// LS Electric XG5000 project: PLC_222
// PLC LSPLC
// module base 0 slot 0: Input/Output Module:XBC-DR30S (DC 24V Input 18 Contacts, Relay Output 12 Contacts)
// module base 0 slot 9: Analog Input Module:XBO-AD02A (A/D Voltage/Current Input Type(2 Channels))
// module base 0 slot 10: Analog Input Module:XBO-AD02A (A/D Voltage/Current Input Type(2 Channels))

PROGRAM NewProgram (task: Scan Program)

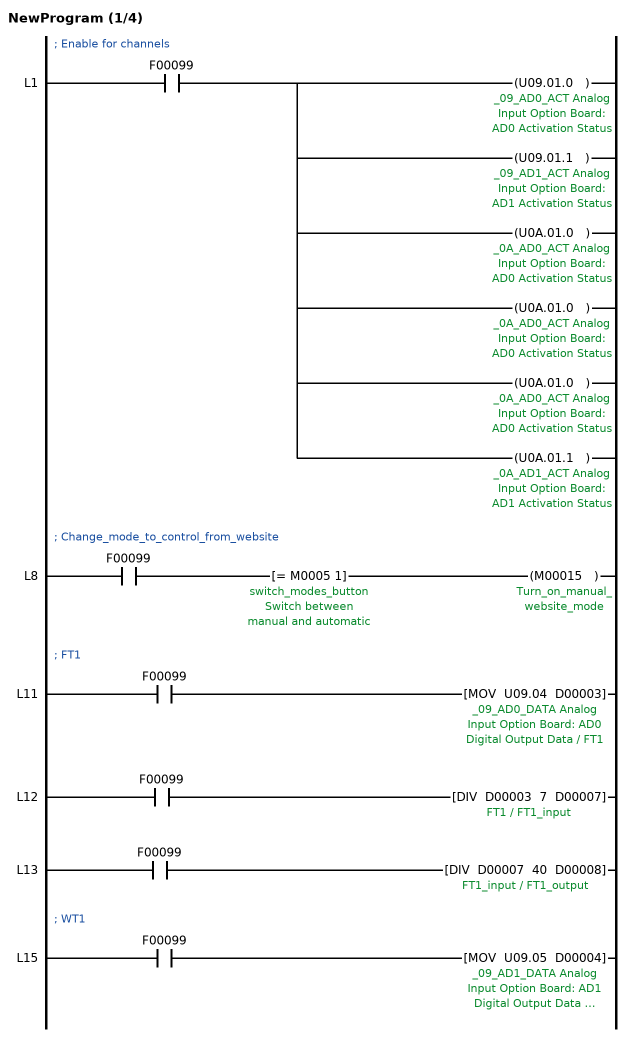
// Enable for channels
; L1
LOAD      F00099
OUT       U09.01.0	// _09_AD0_ACT Analog Input Option Board: AD0 Activation Status
OUT       U09.01.1	// _09_AD1_ACT Analog Input Option Board: AD1 Activation Status
OUT       U0A.01.0	// _0A_AD0_ACT Analog Input Option Board: AD0 Activation Status
OUT       U0A.01.0	// _0A_AD0_ACT Analog Input Option Board: AD0 Activation Status
OUT       U0A.01.0	// _0A_AD0_ACT Analog Input Option Board: AD0 Activation Status
OUT       U0A.01.1	// _0A_AD1_ACT Analog Input Option Board: AD1 Activation Status
// Change_mode_to_control_from_website
; L8
LOAD      F00099
AND=      M0005 1	// switch_modes_button Switch between manual and automatic
OUT       M00015	// Turn_on_manual_website_mode
// FT1
; L11
LOAD      F00099
MOV       U09.04 D00003	// _09_AD0_DATA Analog Input Option Board: AD0 Digital Output Data / FT1
; L12
LOAD      F00099
DIV       D00003 7 D00007	// FT1 / FT1_input
; L13
LOAD      F00099
DIV       D00007 40 D00008	// FT1_input / FT1_output
// WT1
; L15
LOAD      F00099
MOV       U09.05 D00004	// _09_AD1_DATA Analog Input Option Board: AD1 Digital Output Data / WT1_full_range

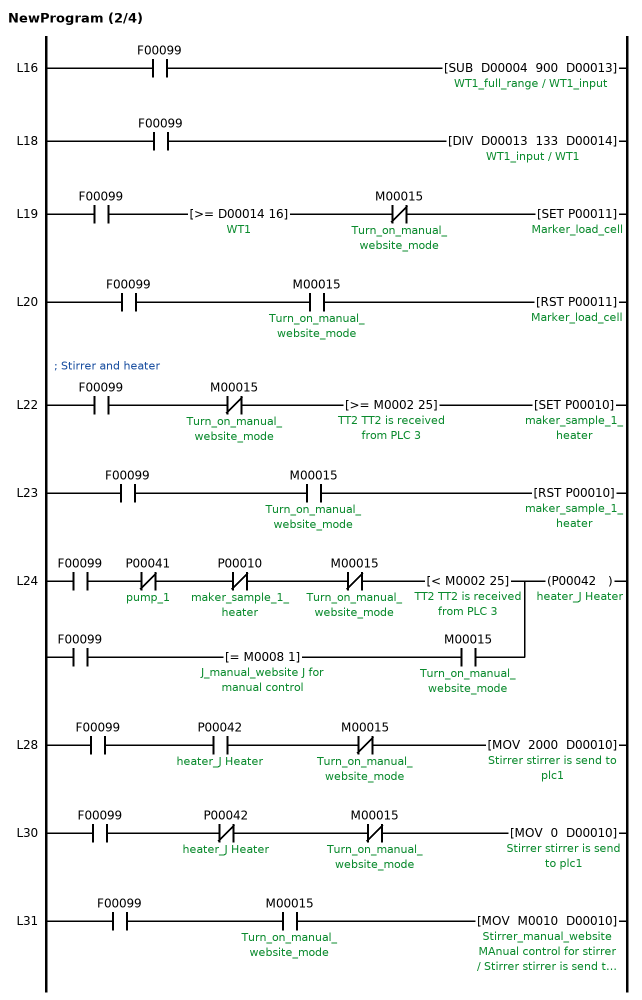
; L16
LOAD      F00099
SUB       D00004 900 D00013	// WT1_full_range / WT1_input
; L18
LOAD      F00099
DIV       D00013 133 D00014	// WT1_input / WT1
; L19
LOAD      F00099
AND>=     D00014 16	// WT1
AND NOT   M00015	// Turn_on_manual_website_mode
SET       P00011	// Marker_load_cell
; L20
LOAD      F00099
AND       M00015	// Turn_on_manual_website_mode
RST       P00011	// Marker_load_cell
// Stirrer and heater
; L22
LOAD      F00099
AND NOT   M00015	// Turn_on_manual_website_mode
AND>=     M0002 25	// TT2 TT2 is received from PLC 3
SET       P00010	// maker_sample_1_heater
; L23
LOAD      F00099
AND       M00015	// Turn_on_manual_website_mode
RST       P00010	// maker_sample_1_heater
; L24
LOAD      F00099
AND NOT   P00041	// pump_1
AND NOT   P00010	// maker_sample_1_heater
AND NOT   M00015	// Turn_on_manual_website_mode
AND<      M0002 25	// TT2 TT2 is received from PLC 3
LOAD      F00099
AND=      M0008 1	// J_manual_website J for manual control
AND       M00015	// Turn_on_manual_website_mode
OR LOAD
OUT       P00042	// heater_J Heater
; L28
LOAD      F00099
AND       P00042	// heater_J Heater
AND NOT   M00015	// Turn_on_manual_website_mode
MOV       2000 D00010	// Stirrer stirrer is send to plc1
; L30
LOAD      F00099
AND NOT   P00042	// heater_J Heater
AND NOT   M00015	// Turn_on_manual_website_mode
MOV       0 D00010	// Stirrer stirrer is send to plc1
; L31
LOAD      F00099
AND       M00015	// Turn_on_manual_website_mode
MOV       M0010 D00010	// Stirrer_manual_website MAnual control for stirrer  / Stirrer stirrer is send to plc1

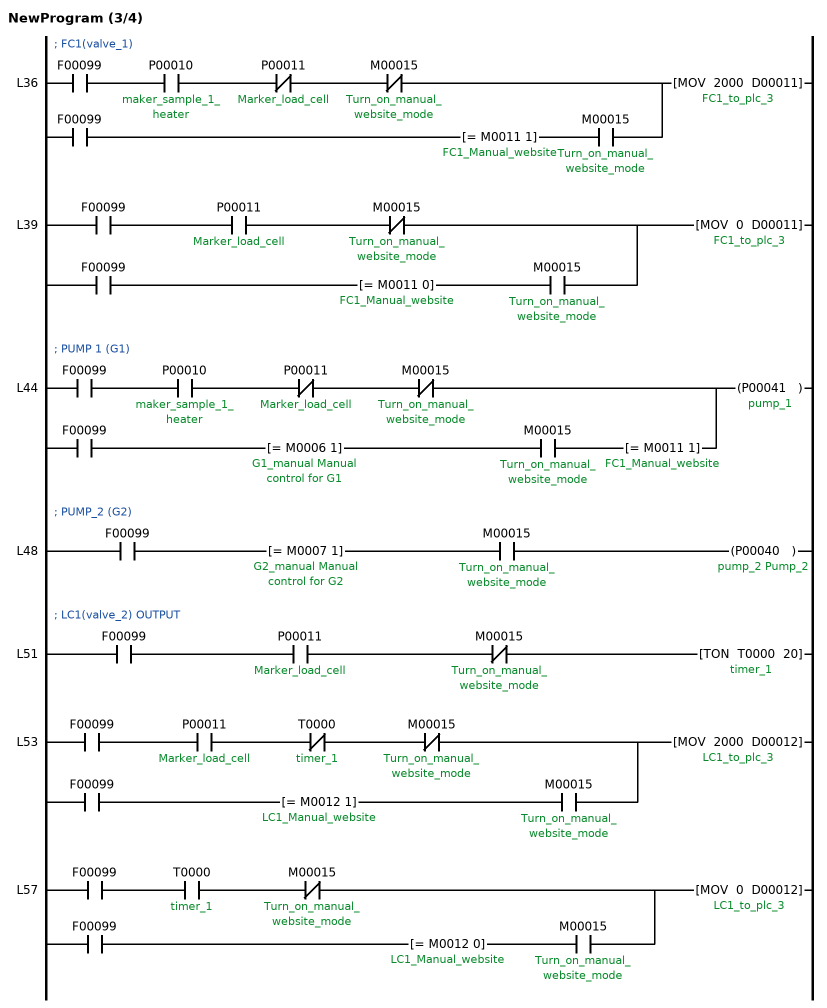
// FC1(valve_1)
; L36
LOAD      F00099
AND       P00010	// maker_sample_1_heater
AND NOT   P00011	// Marker_load_cell
AND NOT   M00015	// Turn_on_manual_website_mode
LOAD      F00099
AND=      M0011 1	// FC1_Manual_website
AND       M00015	// Turn_on_manual_website_mode
OR LOAD
MOV       2000 D00011	// FC1_to_plc_3
; L39
LOAD      F00099
AND       P00011	// Marker_load_cell
AND NOT   M00015	// Turn_on_manual_website_mode
LOAD      F00099
AND=      M0011 0	// FC1_Manual_website
AND       M00015	// Turn_on_manual_website_mode
OR LOAD
MOV       0 D00011	// FC1_to_plc_3
// PUMP 1 (G1)
; L44
LOAD      F00099
AND       P00010	// maker_sample_1_heater
AND NOT   P00011	// Marker_load_cell
AND NOT   M00015	// Turn_on_manual_website_mode
LOAD      F00099
AND=      M0006 1	// G1_manual Manual control for G1
AND       M00015	// Turn_on_manual_website_mode
AND=      M0011 1	// FC1_Manual_website
OR LOAD
OUT       P00041	// pump_1
// PUMP_2 (G2)
; L48
LOAD      F00099
AND=      M0007 1	// G2_manual Manual control for G2
AND       M00015	// Turn_on_manual_website_mode
OUT       P00040	// pump_2 Pump_2
// LC1(valve_2) OUTPUT 
; L51
LOAD      F00099
AND       P00011	// Marker_load_cell
AND NOT   M00015	// Turn_on_manual_website_mode
TON       T0000 20	// timer_1
; L53
LOAD      F00099
AND       P00011	// Marker_load_cell
AND NOT   T0000	// timer_1
AND NOT   M00015	// Turn_on_manual_website_mode
LOAD      F00099
AND=      M0012 1	// LC1_Manual_website
AND       M00015	// Turn_on_manual_website_mode
OR LOAD
MOV       2000 D00012	// LC1_to_plc_3
; L57
LOAD      F00099
AND       T0000	// timer_1
AND NOT   M00015	// Turn_on_manual_website_mode
LOAD      F00099
AND=      M0012 0	// LC1_Manual_website
AND       M00015	// Turn_on_manual_website_mode
OR LOAD
MOV       0 D00012	// LC1_to_plc_3

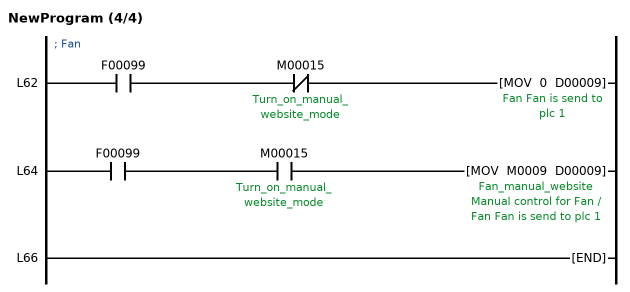
// Fan
; L62
LOAD      F00099
AND NOT   M00015	// Turn_on_manual_website_mode
MOV       0 D00009	// Fan Fan is send to plc 1
; L64
LOAD      F00099
AND       M00015	// Turn_on_manual_website_mode
MOV       M0009 D00009	// Fan_manual_website Manual control for Fan / Fan Fan is send to plc 1
; L66
END

VARIABLES AND COMMENTS (devices not used above)
D00002	WORD	CE1
D00001	WORD	CE1_input
D00011.0	BIT	FC1 // valve_1 is send to plc 3
D00005	WORD	g1_input
C0004	BIT/WORD	heater_2off
D00012.0	BIT	LC1 // valve_2 is send to plc3
M0003	WORD	LT1 // LT1 is received from PLC 3
P00012	BIT	marker_pump2_on
M0014	WORD	marker_stirrer
P00003	BIT	PA1
P00004	BIT	PA2
T0003	BIT/WORD	Pump_2_timer
K00003	BIT	reset_heater_After3samples
K00001	BIT	sampe2_WT1
K00000	BIT	Second_sample
M0001	WORD	ST1 // ST1  is received from PLC 1 
T0001	BIT/WORD	timer_2
M0000	WORD	TT1 // TT1  is received from PLC 1
C0000	BIT/WORD	WT1_counter
C0003	BIT/WORD	WT1_counter_2